FUNCTION_BLOCK FB_PD4
VAR_INPUT
	PD4_IN 			: ST_PD4_IN;
	Enable 			: BOOL;
	ErrorReset 		: BOOL;
	TargetVelocity 	: INT;
	TargetPosition	: DINT;			// Check variable type
	Self 			: INT;
END_VAR
VAR_OUTPUT
	PD4_OUT : ST_PD4_OUT;
	Ready 	: BOOL;
	Error	: BOOL;
END_VAR
VAR
//	State 		: DINT;
	State		: (DEFAULT, INIT, SWITCH_ON_DISABLED, READY_TO_SWITCH_ON, SWITCHED_ON, OPERATION_ENABLED, ERROR);
	PrevState 	: (DEFAULT, INIT, SWITCH_ON_DISABLED, READY_TO_SWITCH_ON, SWITCHED_ON, OPERATION_ENABLED, ERROR);
	StateEntry 	: BOOL;
	Homed		: BOOL;
END_VAR

// POWER FSM State Machine for EtherCAT PD4 Control

IF State <> PrevState THEN
	StateEntry := TRUE;
	PrevState := State;
ELSE
	StateEntry := FALSE;
END_IF

CASE State OF
	DEFAULT:
		State := INIT;
		
	INIT:
		Ready := FALSE;
		PD4_OUT.ControlWord := PD4ControlWord.PulseInhibit;
		PD4_OUT.Polarity := PD4Polarity.Positive;
		
		PD4_OUT.OperationMode := PD4OperationMode.HomingMode;
		PD4_OUT.HomingMethod := 35;									// Zero at current position
		PD4_OUT.ControlWord := PD4ControlWord.StartHoming;
		
		IF PD4_IN.ActualPosition = 0 THEN
			SetMode(PD4OperationMode.ProfilePositionMode);
			SetAbsoluteMotion();
//			SetMode(PD4OperationMode.VelocityMode);
			State := SWITCH_ON_DISABLED;
		END_IF

	SWITCH_ON_DISABLED:
		IF StateEntry THEN
			PD4_OUT.ControlWord := PD4ControlWord.PulseInhibit;
			PD4_OUT.TargetVelocity := 0;
		END_IF
		
		IF ((PD4_IN.StatusWord AND PD4StatusWord.SwitchOnDisabled) = PD4StatusWord.SwitchOnDisabled) THEN
			PD4_OUT.ControlWord := PD4ControlWord.Shutdown;
			State := READY_TO_SWITCH_ON;
		END_IF
		
	READY_TO_SWITCH_ON:
		IF ((PD4_IN.StatusWord AND PD4StatusWOrd.ReadyToSwitchOn) = PD4StatusWOrd.ReadyToSwitchOn) THEN
			PD4_OUT.ControlWord := PD4ControlWord.SwitchOn;
			State := SWITCHED_ON;
		END_IF
		
	SWITCHED_ON:
		IF StateEntry THEN
			Ready := TRUE;
		END_IF
		
		IF (((PD4_IN.StatusWord AND PD4StatusWOrd.SwitchedOn) = PD4StatusWOrd.SwitchedOn) AND Enable) THEN
			PD4_OUT.TargetPosition := PD4_IN.ActualPosition;
			PD4_OUT.ControlWord := PD4ControlWord.EnableOperation;
			State := OPERATION_ENABLED;
		END_IF
		
	OPERATION_ENABLED:
		IF StateEntry THEN
			PD4_OUT.TargetPosition := PD4_IN.ActualPosition;
			TargetPosition := PD4_IN.ActualPosition;
		END_IF
		
		PD4_OUT.TargetPosition := TargetPosition;
		ToggleMoveBit();
//		PD4_OUT.TargetVelocity := TargetVelocity;	
		
		IF NOT Enable THEN
//			PD4_OUT.TargetVelocity := 0;
			PD4_OUT.TargetPosition := PD4_IN.ActualPosition;
			PD4_OUT.ControlWord := PD4ControlWord.DisableOperation;
			State := SWITCHED_ON;
		END_IF
		
	ERROR:
		IF StateEntry THEN
			Ready := FALSE;
			Error := TRUE;	
		END_IF
		
		IF ErrorReset THEN
			PD4_OUT.ControlWord := PD4ControlWord.FaultReset;
			IF ((PD4_IN.StatusWord AND PD4StatusWOrd.Fault) = 0) THEN
				Error := FALSE;
				State := SWITCH_ON_DISABLED;
			END_IF
		END_IF
END_CASE

IF ((PD4_IN.StatusWord AND PD4StatusWord.Fault) = PD4StatusWord.Fault) THEN
	State := ERROR;
END_IF

METHOD SetAbsoluteMotion : BOOL
VAR_INPUT
END_VAR
PD4_OUT.ControlWord := PD4_OUT.ControlWord OR PD4ControlWord.AbsoluteMotion;
END_METHOD

METHOD SetMaxCurrent : BOOL
VAR_INPUT
END_VAR
END_METHOD

METHOD SetMode : BOOL
VAR_INPUT
	OperationMode	: PD4OperationMode;
END_VAR
PD4_OUT.OperationMode := OperationMode;
PD4_OUT.SubmodeSelect := 1;
END_METHOD

METHOD SetMotionProfile : BOOL
VAR_INPUT
	Velocity 	: UDINT;
	Accel 		: UDINT;
	Decel 		: UDINT;
END_VAR
PD4_OUT.ProfileVelocity := Velocity;
PD4_OUT.Accel := Accel;
PD4_OUT.Decel := Decel;
END_METHOD

METHOD ToggleMoveBit : BOOL
VAR_INPUT
END_VAR
IF (PD4_OUT.ControlWord AND PD4ControlWord.StartMove) = PD4ControlWord.StartMove THEN
	PD4_OUT.ControlWord := (PD4_OUT.ControlWord AND (NOT PD4ControlWord.StartMove));
ELSE
	PD4_OUT.ControlWord := (PD4_OUT.ControlWord OR PD4ControlWord.StartMove);
END_IF
END_METHOD

END_FUNCTION_BLOCK

(* stored: Version 1.1.0.1, ProductVersion 3.1.4024.12
   POU FB_PD4: Id {e09cee4c-9330-4994-9354-d4a609a75133}, SpecialFunc None
   Method SetAbsoluteMotion: Id {b00f98ed-136b-4e21-9922-598b4502a478}
   Method SetMaxCurrent: Id {d71f4290-7d0f-46e0-b5da-4ed562328b8c}
   Method SetMode: Id {dc242788-6c1e-42b7-8aef-54f3132ad46b}
   Method SetMotionProfile: Id {22327d2a-0c20-4efc-a559-247f210439c1}
   Method ToggleMoveBit: Id {778237c8-e827-42a5-bdd7-6ccd9a52a9fb} *)
